# EPICS IOC start-up script: test/startup/st.mcu007-PTP-utgard.iocsh
require EthercatMC,USER

epicsEnvSet("MOTOR_PORT",    "$(SM_MOTOR_PORT=MCU1)")

epicsEnvSet("IPADDR",        "$(SM_IPADDR=172.30.244.150)")
epicsEnvSet("IPPORT",        "$(SM_IPPORT=48898)")
epicsEnvSet("ASYN_PORT",     "$(SM_ASYN_PORT=MC_CPU1)")
epicsEnvSet("PREFIX",        "$(SM_PREFIX=LabS-MCAG:MC-MCU-07:)")
epicsEnvSet("PREC",          "$(SM_PREC=3)")
epicsEnvSet("SM_NOAXES",     "1")
epicsEnvSet("ECM_OPTIONS",   "adsPort=852;amsNetIdRemote=192.168.88.57.1.1;amsNetIdLocal=172.30.244.38.1.1"

< ethercatmcController.iocsh
< ethercatmcEL6688-PTP.iocsh
< ethercatmcEL6688-ExtSync.iocsh

#
# Axis 1
#
epicsEnvSet("AXISCONFIG",    "")
epicsEnvSet("MOTOR_NAME",    "$(SM_MOTOR_NAME=m1)")
epicsEnvSet("AXIS_NO",       "$(SM_AXIS_NO=1)")
epicsEnvSet("DESC",          "$(SM_DESC=DESC)")
epicsEnvSet("EGU",           "$(SM_EGU=EGU)")
< ethercatmcIndexerAxis.iocsh
< ethercatmcAxisdebug.iocsh
< ethercatmcAxishome.iocsh

# Raw steps and velocity
< ethercatmcRawMtrEnc.iocsh

# Predefined Positions
epicsEnvSet("NVL",           "")
epicsEnvSet("EGU",           "")
< ethercatmcDefPos.iocsh
< ethercatmcRawMtrEnc.iocsh

#####################################################
# EL1252, first channel, CHNO == 0
epicsEnvSet("CHNO",     "0")
< ethercatmcEL1252-OneChannel.iocsh

#####################################################
# PTP with ExtSync
< ethercatmcEL6688-PTP.iocsh
< ethercatmcEL6688-ExtSync.iocsh

#
# Start polling, values are in millisconds
#
epicsEnvSet("MOVINGPOLLPERIOD", "50")
epicsEnvSet("IDLEPOLLPERIOD",   "100")
ethercatmcStartPoller("$(MOTOR_PORT)", "$(MOVINGPOLLPERIOD)", "$(IDLEPOLLPERIOD)")
